FUNCTION_BLOCK FB_Sensor IMPLEMENTS I_Sensor
VAR_INPUT
END_VAR
VAR_OUTPUT
END_VAR
VAR
	_Calibrar 		: BOOL;
	Valor			: INT;
	_Temperatura 	: REAL;
	_Consigna       : REAL;

END_VAR

PROPERTY Calibrado : BOOL
GET
Calibrado := _Calibrar;
END_GET
END_PROPERTY


METHOD Calibrar
THIS^._Calibrar := TRUE;
END_METHOD

PROPERTY Consigna : REAL
SET
THIS^._Consigna := Consigna;
END_SET
END_PROPERTY

METHOD Descalibrar
THIS^._Calibrar := FALSE;
END_METHOD


METHOD LeerValor : INT
LeerValor := Valor;
END_METHOD


PROPERTY Temperatura : REAL
GET
Temperatura := THIS^._Temperatura;
END_GET
END_PROPERTY

END_FUNCTION_BLOCK

(* stored: Version 1.1.0.1, ProductVersion 3.1.4024.12
   POU FB_Sensor: Id {053f071d-af09-4910-ba64-dff4b8a61f15}, SpecialFunc None
   Property Calibrado: Id {9d63c4dd-53c9-4ddb-b6cb-5a12d007b478}
   Get Get: Id {59593ab4-c379-4315-80ec-ad3b2aa0747c}
   Method Calibrar: Id {80ffb7cf-22c3-401e-9cfe-ec22fdb72363}
   Property Consigna: Id {f56818bf-5b52-486f-b05e-793e3f037a4e}
   Set Set: Id {c1bf984f-d2f9-4644-bcd0-79dd31ba8d47}
   Method Descalibrar: Id {e0ba46fa-e6d0-4727-9e3a-1c54143318aa}
   Method LeerValor: Id {e4da853c-2a44-4d03-8c4b-078f6523d9e5}
   Property Temperatura: Id {d77617b0-0e98-4ddc-aa4b-491e7ea2847c}
   Get Get: Id {9318b208-42bd-4cd7-9273-921fea2b06e5} *)
